VAR_GLOBAL
	WaySectionGap		: LREAL := 110.0;
	WaitingAbsPosition	: LREAL := 950;
	
	Startposition		: ARRAY[1..AxCnt] OF LREAL; // positionen, in denen sich die mover vor couple einfinden
END_VAR

(* stored: Version 1.1.0.1, ProductVersion 3.1.0.25
   GVL SkillHandleConstants: Id {ecbb643c-e846-4509-95f4-2085deb32320} *)
